INTERFACE I_LightDimmable EXTENDS I_LightBase

PROPERTY Brightness : USINT
GET
END_GET
SET
END_SET
END_PROPERTY

END_INTERFACE

(* stored: Version 1.1.0.1, ProductVersion 3.1.4024.12
   Itf I_LightDimmable: Id {88a95757-277b-49ff-95f3-abd80b37f3b7}
   Property Brightness: Id {622b1b12-8ea9-41ce-a6ee-84ff45cd706d}
   Get Get: Id {be354563-f0ab-49d8-9e60-c53b1b49b282}
   Set Set: Id {0ff90000-552a-4d06-b039-b26c2ff73e94} *)
